(* IEC 61131-3 sources: io/test/Output, 7 files *)

(* ---- DintOutputTest.st ---- *)
USING Simatic.Ax.IO.Output;
USING AxUnit;

NAMESPACE Simatic.Ax.IO.Output.Test

    /// Test fixture for DintOutput class
    /// Verifies double integer (DINT) output functionality including:
    /// - Setting output values via SetValue()
    /// - Writing values cyclically via WriteCyclic()
    /// - Change detection via HasChanged()
    {TestFixture}
    CLASS TestDIntOutputSetValueClass
        VAR
            o : DIntOutput;  // Test object for DintOutput
            oHasChanged : DIntOutput;  // Test object for change detection
        END_VAR

        /// Parameterized test for setting and writing DINT output values
        /// Verifies SetValue() and WriteCyclic() work correctly
        {Test(value := DINT#0, actual := DINT#0)}
        {Test(value := DINT#1, actual := DINT#1)}
        METHOD PUBLIC TestOutputSetValue
            VAR_INPUT
                value : DINT;
                actual : DINT;
            END_VAR
            VAR_TEMP
                _expect : DINT;
            END_VAR

            o.SetValue(value := value);
            o.WriteCyclic(Q => _expect);
            Assert.Equal(expected := _expect, actual := actual);
        END_METHOD

        /// Test change detection functionality
        /// Verifies HasChanged() returns TRUE after value changes
        {Test}
        METHOD PUBLIC TestOutputHasChanged
            VAR_TEMP
                value : DINT;
            END_VAR
            Assert.Equal(FALSE, oHasChanged.HasChanged());
            oHasChanged.SetValue(value := DINT#1);
            oHasChanged.WriteCyclic(Q => value);
            Assert.Equal(TRUE, oHasChanged.HasChanged());
        END_METHOD
    END_CLASS
END_NAMESPACE

(* ---- DWordOutputTest.st ---- *)
USING Simatic.Ax.IO.Output;
USING AxUnit;

NAMESPACE Simatic.Ax.IO.Output.Test

    /// Test fixture for DWordOutput class
    /// Verifies double word (DWORD) output functionality including:
    /// - Setting output values via SetValue()
    /// - Writing values cyclically via WriteCyclic()
    /// - Change detection via HasChanged()
    {TestFixture}
    CLASS TestDWordOutputSetValueClass
        VAR
            o : DWordOutput;  // Test object for DWordOutput
            oHasChanged : DWordOutput;  // Test object for change detection
        END_VAR

        /// Parameterized test for setting and writing DWORD output values
        /// Verifies SetValue() and WriteCyclic() work correctly
        {Test(value := DWORD#16#0, actual := DWORD#16#0)}
        {Test(value := DWORD#16#1, actual := DWORD#16#1)}
        METHOD PUBLIC TestOutputSetValue
            VAR_INPUT
                value : DWORD;
                actual : DWORD;
            END_VAR
            VAR_TEMP
                _expect : DWORD;
            END_VAR

            o.SetValue(value := value);
            o.WriteCyclic(Q => _expect);
            Assert.Equal(expected := _expect, actual := actual);
        END_METHOD

        /// Test change detection functionality
        /// Verifies HasChanged() returns TRUE after value changes
        {Test}
        METHOD PUBLIC TestOutputHasChanged
            VAR_TEMP
                value : DWORD;
            END_VAR
            Assert.Equal(FALSE, oHasChanged.HasChanged());
            oHasChanged.SetValue(value := DWORD#1);
            oHasChanged.WriteCyclic(Q => value);
            Assert.Equal(TRUE, oHasChanged.HasChanged());
        END_METHOD
    END_CLASS
END_NAMESPACE

(* ---- IntOutputTest.st ---- *)
USING Simatic.Ax.IO.Output;
USING AxUnit;

NAMESPACE Simatic.Ax.IO.Output.Test

    /// Test fixture for IntOutput class
    /// Verifies integer (INT) output functionality including:
    /// - Setting output values via SetValue()
    /// - Writing values cyclically via WriteCyclic()
    /// - Change detection via HasChanged()
    {TestFixture}
    CLASS TestIntOutputSetValueClass
        VAR
            o : IntOutput;  // Test object for IntOutput
            oHasChanged : IntOutput;  // Test object for change detection
        END_VAR

        /// Parameterized test for setting and writing INT output values
        /// Verifies SetValue() and WriteCyclic() work correctly
        {Test(value := 0, actual := 0)}
        {Test(value := 1, actual := 1)}
        METHOD PUBLIC TestOutputSetValue
            VAR_INPUT
                value : INT;
                actual : INT;
            END_VAR
            VAR_TEMP
                _expect : INT;
            END_VAR

            o.SetValue(value := value);
            o.WriteCyclic(Q => _expect);
            Assert.Equal(expected := _expect, actual := actual);
        END_METHOD

        /// Test change detection functionality
        /// Verifies HasChanged() returns TRUE after value changes
        {Test}
        METHOD PUBLIC TestOutputHasChanged
            VAR_TEMP
                value : INT;
            END_VAR
            Assert.Equal(FALSE, oHasChanged.HasChanged());
            oHasChanged.SetValue(value := 1);
            oHasChanged.WriteCyclic(Q => value);
            Assert.Equal(TRUE, oHasChanged.HasChanged());
        END_METHOD
    END_CLASS
END_NAMESPACE

(* ---- LintOutputTest.st ---- *)
USING Simatic.Ax.IO.Output;
USING AxUnit;

NAMESPACE Simatic.Ax.IO.Output.Test

    /// Test fixture for LIntOutput class
    /// Verifies long integer (LINT) output functionality including:
    /// - Setting output values via SetValue()
    /// - Writing values cyclically via WriteCyclic()
    /// - Change detection via HasChanged()
    {TestFixture}
    CLASS TestLIntOutputSetValueClass
        VAR
            o : LIntOutput;  // Test object for LIntOutput
            oHasChanged : LIntOutput;  // Test object for change detection
        END_VAR

        /// Parameterized test for setting and writing LINT output values
        /// Verifies SetValue() and WriteCyclic() work correctly
        {Test(value := LINT#0, actual := LINT#0)}
        {Test(value := LINT#1, actual := LINT#1)}
        METHOD PUBLIC TestOutputSetValue
            VAR_INPUT
                value : LINT;
                actual : LINT;
            END_VAR
            VAR_TEMP
                _expect : LINT;
            END_VAR

            o.SetValue(value := value);
            o.WriteCyclic(Q => _expect);
            Assert.Equal(expected := _expect, actual := actual);
        END_METHOD

        /// Test change detection functionality
        /// Verifies HasChanged() returns TRUE after value changes
        {Test}
        METHOD PUBLIC TestOutputHasChanged
            VAR_TEMP
                value : LINT;
            END_VAR
            Assert.Equal(FALSE, oHasChanged.HasChanged());
            oHasChanged.SetValue(value := LINT#1);
            oHasChanged.WriteCyclic(Q => value);
            Assert.Equal(TRUE, oHasChanged.HasChanged());
        END_METHOD
    END_CLASS
END_NAMESPACE

(* ---- LRealTest.st ---- *)
USING Simatic.Ax.IO.Output;
USING AxUnit;

NAMESPACE Simatic.Ax.IO.Output.Test

    /// Test fixture for LRealOutput class
    /// Verifies long real (LREAL) double precision floating-point output functionality including:
    /// - Setting output values via SetValue()
    /// - Writing values cyclically via WriteCyclic() as LWORD bit pattern
    /// - Change detection via HasChanged()
    {TestFixture}
    CLASS TestLRealOutputSetValueClass
        VAR
            o : LRealOutput;  // Test object for LRealOutput
            oHasChanged : LRealOutput;  // Test object for change detection
        END_VAR

        /// Parameterized test for setting and writing LREAL output values
        /// Verifies SetValue() and WriteCyclic() work correctly
        /// Output is converted to LWORD bit pattern for hardware compatibility
        {Test(value := LREAL#0.0, actual := LREAL#0.0)}
        {Test(value := LREAL#1.0, actual := LREAL#1.0)}
        METHOD PUBLIC TestOutputSetValue
            VAR_INPUT
                value : LREAL;
                actual : LREAL;
            END_VAR
            VAR_TEMP
                _expect : LWORD;
            END_VAR

            o.SetValue(value := value);
            o.WriteCyclic(Q => _expect);
            Assert.Equal(expected := _expect, actual := TO_LWORD(actual));
        END_METHOD

        /// Test change detection functionality
        /// Verifies HasChanged() returns TRUE after value changes
        {Test}
        METHOD PUBLIC TestOutputHasChanged
            VAR_TEMP
                value : LWORD;
            END_VAR
            Assert.Equal(FALSE, oHasChanged.HasChanged());
            oHasChanged.SetValue(value := LREAL#1.0);
            oHasChanged.WriteCyclic(Q => value);
            Assert.Equal(TRUE, oHasChanged.HasChanged());
        END_METHOD
    END_CLASS
END_NAMESPACE

(* ---- RealOutputTest.st ---- *)
USING Simatic.Ax.IO.Output;
USING AxUnit;

NAMESPACE Simatic.Ax.IO.Output.Test

    /// Test fixture for RealOutput class
    /// Verifies real (REAL) floating-point output functionality including:
    /// - Setting output values via SetValue()
    /// - Writing values cyclically via WriteCyclic() as DWORD bit pattern
    /// - Change detection via HasChanged()
    {TestFixture}
    CLASS TestRealOutputSetValueClass
        VAR
            o : RealOutput;  // Test object for RealOutput
            oHasChanged : RealOutput;  // Test object for change detection
        END_VAR

        /// Parameterized test for setting and writing REAL output values
        /// Verifies SetValue() and WriteCyclic() work correctly
        /// Output is converted to DWORD bit pattern for hardware compatibility
        {Test(value := REAL#0.0, actual := REAL#0.0)}
        {Test(value := REAL#1.0, actual := REAL#1.0)}
        METHOD PUBLIC TestWordOutputSetValue
            VAR_INPUT
                value : REAL;
                actual : REAL;
            END_VAR
            VAR_TEMP
                _expect : DWORD;
            END_VAR

            o.SetValue(value := value);
            o.WriteCyclic(Q => _expect);
            Assert.Equal(expected := _expect, actual := TO_DWORD(actual));
        END_METHOD

        /// Test change detection functionality
        /// Verifies HasChanged() returns TRUE after value changes
        {Test}
        METHOD PUBLIC TestRealOutputHasChanged
            VAR_TEMP
                value : DWORD;
            END_VAR
            Assert.Equal(FALSE, oHasChanged.HasChanged());
            oHasChanged.SetValue(value := REAL#1.0);
            oHasChanged.WriteCyclic(Q => value);
            Assert.Equal(TRUE, oHasChanged.HasChanged());
        END_METHOD
    END_CLASS
END_NAMESPACE

(* ---- WordOutputTest.st ---- *)
USING Simatic.Ax.IO.Output;
USING AxUnit;

NAMESPACE Simatic.Ax.IO.Output.Test

    /// Test fixture for WordOutput class
    /// Verifies word (WORD) output functionality including:
    /// - Setting output values via SetValue()
    /// - Writing values cyclically via WriteCyclic()
    /// - Change detection via HasChanged()
    {TestFixture}
    CLASS TestWordOutputSetValueClass
        VAR
            o : WordOutput;  // Test object for WordOutput
            oHasChanged : WordOutput;  // Test object for change detection
        END_VAR

        /// Parameterized test for setting and writing WORD output values
        /// Verifies SetValue() and WriteCyclic() work correctly
        {Test(value := WORD#16#0, actual := WORD#16#0)}
        {Test(value := WORD#16#1, actual := WORD#16#1)}
        METHOD PUBLIC TestOutputSetValue
            VAR_INPUT
                value : WORD;
                actual : WORD;
            END_VAR
            VAR_TEMP
                _expect : WORD;
            END_VAR

            o.SetValue(value := value);
            o.WriteCyclic(Q => _expect);
            Assert.Equal(expected := _expect, actual := actual);
        END_METHOD

        /// Test change detection functionality
        /// Verifies HasChanged() returns TRUE after value changes
        {Test}
        METHOD PUBLIC TestOutputHasChanged
            VAR_TEMP
                value : Word;
            END_VAR
            Assert.Equal(FALSE, oHasChanged.HasChanged());
            oHasChanged.SetValue(value := WORD#1);
            oHasChanged.WriteCyclic(Q => value);
            Assert.Equal(TRUE, oHasChanged.HasChanged());
        END_METHOD
    END_CLASS
END_NAMESPACE
